TYPE (* A Template for a Data Type *)
  (* Description: Copyright (c) 2026 Sichuan Qunyuan Technology Co., Ltd. This program and the accompanying materials are made available under the terms of the Eclipse Public License 2.0 which is available at https://www.eclipse.org/legal/epl-2.0/ SPDX-License-Identifier: EPL-2.0 *)
  (* Version 1.0, 2026-04-10, Zijun Tang *)
  PACKAGE eclipse4diac::io::ethercat;
  ECDeviceConfig : STRUCT
    Alias : UINT;
    Position : UINT;
    VendorId : UDINT;
    ProductCode : UDINT;
  END_STRUCT;
END_TYPE
